FUNCTION_BLOCK INFO_WRAPPER
  {SET_ATTRIBUTE(OpcUa, METHOD)}
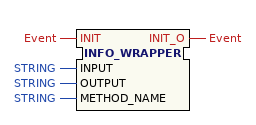
  EVENT_INPUT
    INIT;
  END_EVENT
  EVENT_OUTPUT
    INIT_O;
  END_EVENT
  VAR_INPUT
    INPUT : STRING; {SET_ATTRIBUTE(OpcUa, Constant.INIT)}
    OUTPUT : STRING; {SET_ATTRIBUTE(OpcUa, Constant.INIT)}
    METHOD_NAME : STRING; {SET_ATTRIBUTE(OpcUa, Constant.INIT)}
  END_VAR
END_FUNCTION_BLOCK
